# EPICS autosave request: ioc/autoSaveRestore/ramp1Menu.req
file configMenu.req P=$(P), CONFIG=$(CONFIG)
file rampSetting.req P=$(P), S=ramp1
